PROGRAM MAIN
VAR
	b1: BOOL;
	b2: BOOL;
	c1: BOOL;

END_VAR

END_PROGRAM

(* stored: Version 1.1.0.1, ProductVersion 3.1.4024.11
   POU MAIN: Id {acfcde57-02b8-4fc3-846d-8c496d7e560d}, SpecialFunc None *)
